FUNCTION_BLOCK Utilities (* Composite Function Block Type *)
  (* Standard: 61499-2 *)
  (* Version 0.0, 9/9/2024, SESA685388, Schneider Electric, template *)
  PACKAGE SE.Nereda;
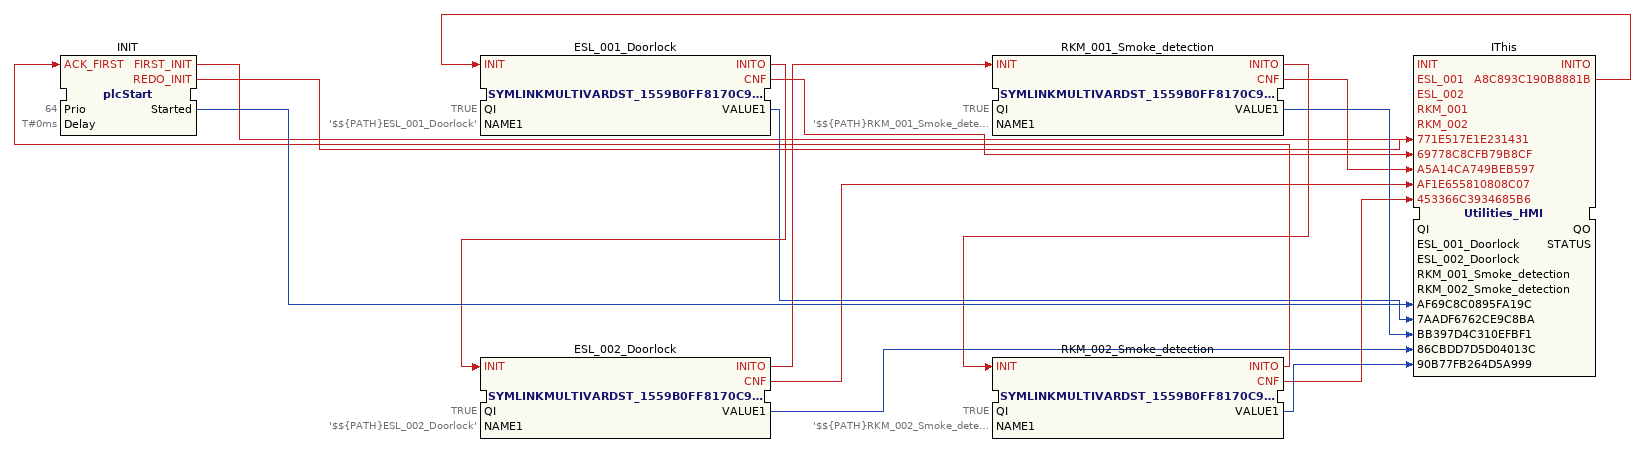
  FBS
    INIT : plcStart(Prio := 64, Delay := T#0ms);
    IThis : Utilities_HMI;
    ESL_001_Doorlock : SYMLINKMULTIVARDST_1559B0FF8170C9BA0(QI := TRUE, NAME1 := '$${PATH}ESL_001_Doorlock'); {SET_ATTRIBUTE(Configuration.GenericFBType.InterfaceParams, Runtime.System#I:=1;VALUE${I$}:BOOL)}
    ESL_002_Doorlock : SYMLINKMULTIVARDST_1559B0FF8170C9BA0(QI := TRUE, NAME1 := '$${PATH}ESL_002_Doorlock'); {SET_ATTRIBUTE(Configuration.GenericFBType.InterfaceParams, Runtime.System#I:=1;VALUE${I$}:BOOL)}
    RKM_001_Smoke_detection : SYMLINKMULTIVARDST_1559B0FF8170C9BA0(QI := TRUE, NAME1 := '$${PATH}RKM_001_Smoke_detection'); {SET_ATTRIBUTE(Configuration.GenericFBType.InterfaceParams, Runtime.System#I:=1;VALUE${I$}:BOOL)}
    RKM_002_Smoke_detection : SYMLINKMULTIVARDST_1559B0FF8170C9BA0(QI := TRUE, NAME1 := '$${PATH}RKM_002_Smoke_detection'); {SET_ATTRIBUTE(Configuration.GenericFBType.InterfaceParams, Runtime.System#I:=1;VALUE${I$}:BOOL)}
  END_FBS
  EVENT_CONNECTIONS
    ESL_001_Doorlock.INITO TO ESL_002_Doorlock.INIT;
    ESL_002_Doorlock.INITO TO RKM_001_Smoke_detection.INIT;
    RKM_001_Smoke_detection.INITO TO RKM_002_Smoke_detection.INIT;
    RKM_002_Smoke_detection.INITO TO INIT.ACK_FIRST;
    INIT.FIRST_INIT TO IThis.771E517E1E231431;
    INIT.REDO_INIT TO IThis.771E517E1E231431;
    ESL_001_Doorlock.CNF TO IThis.69778C8CFB79B8CF;
    RKM_001_Smoke_detection.CNF TO IThis.A5A14CA749BEB597;
    ESL_002_Doorlock.CNF TO IThis.AF1E655810808C07;
    RKM_002_Smoke_detection.CNF TO IThis.453366C3934685B6;
    IThis.A8C893C190B8881B TO ESL_001_Doorlock.INIT;
  END_CONNECTIONS
  DATA_CONNECTIONS
    INIT.Started TO IThis.AF69C8C0895FA19C;
    ESL_001_Doorlock.VALUE1 TO IThis.7AADF6762CE9C8BA;
    RKM_001_Smoke_detection.VALUE1 TO IThis.BB397D4C310EFBF1;
    ESL_002_Doorlock.VALUE1 TO IThis.86CBDD7D5D04013C;
    RKM_002_Smoke_detection.VALUE1 TO IThis.90B77FB264D5A999;
  END_CONNECTIONS
END_FUNCTION_BLOCK
